FUNCTION_BLOCK basicRevezamento2Motores (* Basic Function Block Type *)
  (* Standard: 61499-2 *)
  (* Version 0.0, 2/10/2026, Schneider Electric, Template *)
  PACKAGE Hidryco.HidrycoLib;
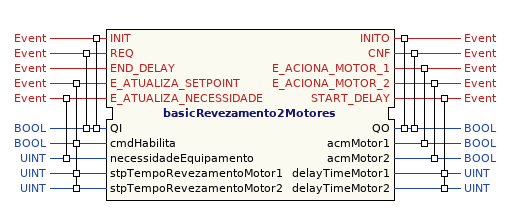
  EVENT_INPUT
    INIT WITH QI; (* Initialization Request *)
    REQ WITH QI; (* Normal Execution Request *)
    END_DELAY;
    E_ATUALIZA_SETPOINT WITH stpTempoRevezamentoMotor1, stpTempoRevezamentoMotor2, cmdHabilita;
    E_ATUALIZA_NECESSIDADE WITH necessidadeEquipamento;
  END_EVENT
  EVENT_OUTPUT
    INITO WITH QO; (* Initialization Confirm *)
    CNF WITH QO; (* Execution Confirmation *)
    E_ACIONA_MOTOR_1 WITH acmMotor1;
    E_ACIONA_MOTOR_2 WITH acmMotor2;
    START_DELAY WITH delayTimeMotor1, delayTimeMotor2;
  END_EVENT
  VAR_INPUT
    QI : BOOL; (* Input event qualifier *)
    cmdHabilita : BOOL;
    necessidadeEquipamento : UINT;
    stpTempoRevezamentoMotor1 : UINT;
    stpTempoRevezamentoMotor2 : UINT;
  END_VAR
  VAR_OUTPUT
    QO : BOOL; (* Output event qualifier *)
    acmMotor1 : BOOL;
    acmMotor2 : BOOL;
    delayTimeMotor1 : UINT;
    delayTimeMotor2 : UINT;
  END_VAR
  VAR
    equipamentoPrincipal : UINT := 1;
  END_VAR
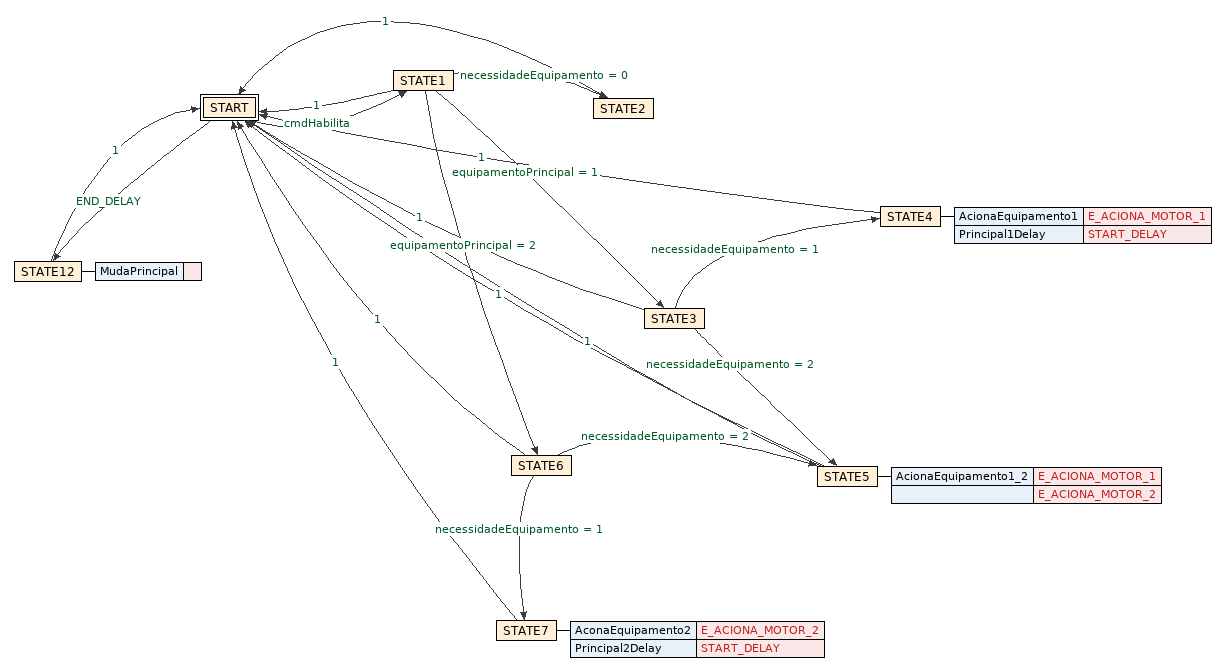
  EC_STATES
    START; (* Initial State *)
    STATE1;
    STATE3;
    STATE2;
    STATE4 : AcionaEquipamento1 -> E_ACIONA_MOTOR_1, Principal1Delay -> START_DELAY;
    STATE5 : AcionaEquipamento1_2 -> E_ACIONA_MOTOR_1, -> E_ACIONA_MOTOR_2;
    STATE6;
    STATE7 : AconaEquipamento2 -> E_ACIONA_MOTOR_2, Principal2Delay -> START_DELAY;
    STATE12 : MudaPrincipal;
  END_STATES
  EC_TRANSITIONS
    START TO STATE1 := cmdHabilita;
    STATE1 TO STATE2 := necessidadeEquipamento = 0;
    STATE2 TO START := 1;
    STATE1 TO STATE3 := equipamentoPrincipal = 1;
    STATE3 TO STATE4 := necessidadeEquipamento = 1;
    STATE4 TO START := 1;
    STATE3 TO STATE5 := necessidadeEquipamento = 2;
    STATE5 TO START := 1;
    STATE3 TO START := 1;
    STATE1 TO STATE6 := equipamentoPrincipal = 2;
    STATE6 TO STATE7 := necessidadeEquipamento = 1;
    STATE7 TO START := 1;
    STATE6 TO START := 1;
    STATE1 TO START := 1;
    START TO STATE12 := END_DELAY;
    STATE12 TO START := 1;
    STATE6 TO STATE5 := necessidadeEquipamento = 2;
    STATE5 TO START := 1;
  END_TRANSITIONS
  ALGORITHM AcionaEquipamento1 IN ST:
acmMotor1 := TRUE;
acmMotor2 := FALSE;
;
  END_ALGORITHM
  ALGORITHM AcionaEquipamento1_2 IN ST:
acmMotor1 := TRUE;
acmMotor2 := TRUE;
;
  END_ALGORITHM
  ALGORITHM AconaEquipamento2 IN ST:
acmMotor1 := FALSE;
acmMotor2 := TRUE;
;
  END_ALGORITHM
  ALGORITHM Principal1Delay IN ST:
delayTimeMotor1 := stpTempoRevezamentoMotor1;
;
  END_ALGORITHM
  ALGORITHM Principal2Delay IN ST:
delayTimeMotor2 := stpTempoRevezamentoMotor2;
;
  END_ALGORITHM
  ALGORITHM MudaPrincipal IN ST:
IF equipamentoPrincipal = 1 THEN
	equipamentoPrincipal := equipamentoPrincipal + 1;
ELSE
	equipamentoPrincipal := 1;
END_IF;
;
  END_ALGORITHM
END_FUNCTION_BLOCK
